PROGRAM F_Gestion_Actionneurs
VAR
	V3V_Bat_Froid_CTA		: Servomoteur_V1;
	Batterie_Elec_CTA		: BatElec;
	Humidificateur			: Humidificateur;
	F_Humi: REAL;
	EF_Humi: BOOL;
	F_BatElec: REAL;
	EF_BatElec: BOOL;
END_VAR
VAR // added by the converter: edge detectors and wires of the graphical bodies
    _w1, _w2 : BOOL;
END_VAR

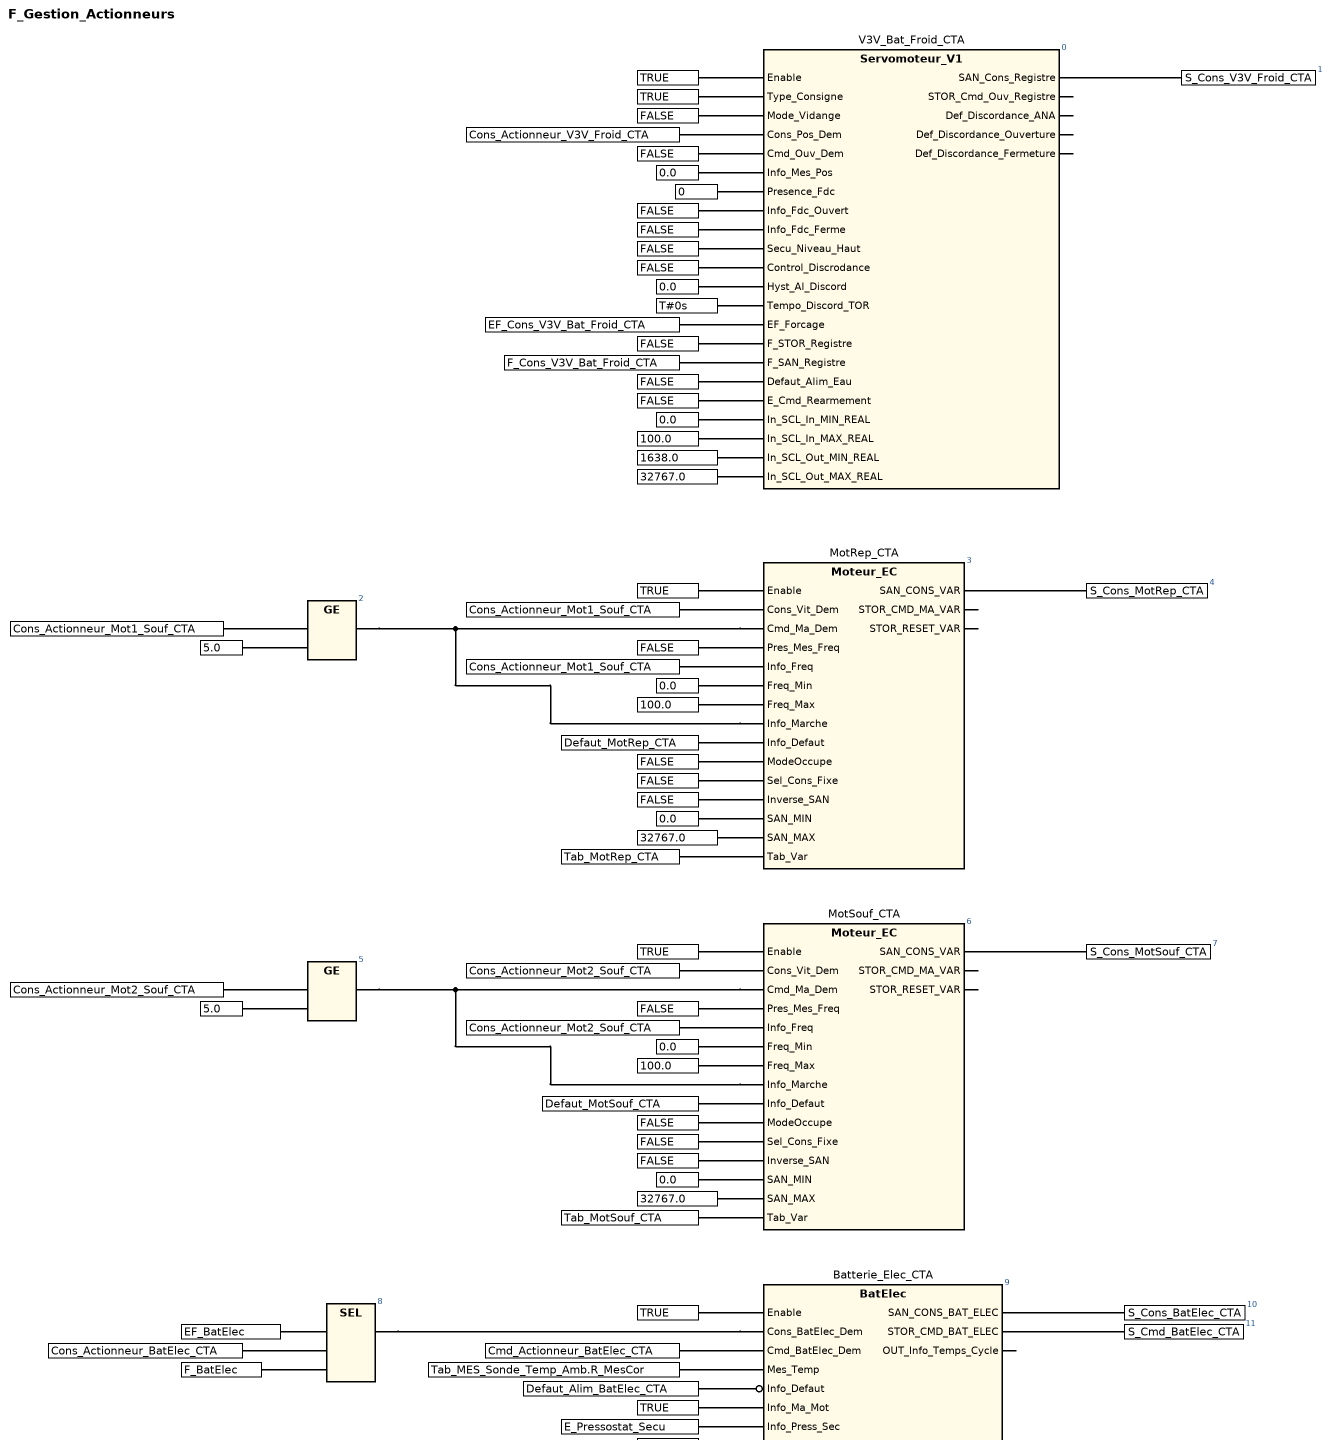
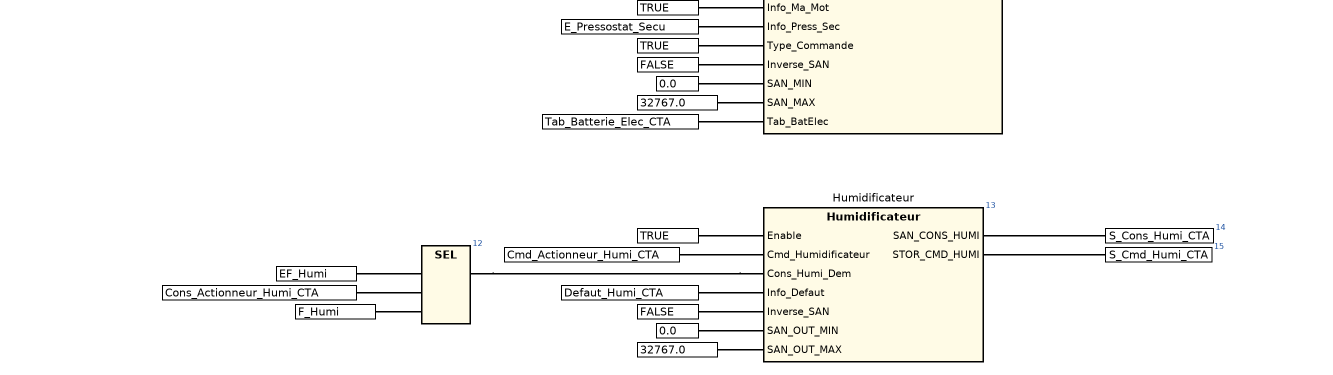
V3V_Bat_Froid_CTA(
    Enable := TRUE,
    Type_Consigne := TRUE,
    Mode_Vidange := FALSE,
    Cons_Pos_Dem := Cons_Actionneur_V3V_Froid_CTA,
    Cmd_Ouv_Dem := FALSE,
    Info_Mes_Pos := 0.0,
    Presence_Fdc := 0,
    Info_Fdc_Ouvert := FALSE,
    Info_Fdc_Ferme := FALSE,
    Secu_Niveau_Haut := FALSE,
    Control_Discrodance := FALSE,
    Hyst_Al_Discord := 0.0,
    Tempo_Discord_TOR := T#0s,
    EF_Forcage := EF_Cons_V3V_Bat_Froid_CTA,
    F_STOR_Registre := FALSE,
    F_SAN_Registre := F_Cons_V3V_Bat_Froid_CTA,
    Defaut_Alim_Eau := FALSE,
    E_Cmd_Rearmement := FALSE,
    In_SCL_In_MIN_REAL := 0.0,
    In_SCL_In_MAX_REAL := 100.0,
    In_SCL_Out_MIN_REAL := 1638.0,
    In_SCL_Out_MAX_REAL := 32767.0); // Servomoteur_V1
S_Cons_V3V_Froid_CTA := V3V_Bat_Froid_CTA.SAN_Cons_Registre;
_w1 := Cons_Actionneur_Mot1_Souf_CTA >= 5.0;
MotRep_CTA(
    Enable := TRUE,
    Cons_Vit_Dem := Cons_Actionneur_Mot1_Souf_CTA,
    Cmd_Ma_Dem := _w1,
    Pres_Mes_Freq := FALSE,
    Info_Freq := Cons_Actionneur_Mot1_Souf_CTA,
    Freq_Min := 0.0,
    Freq_Max := 100.0,
    Info_Marche := _w1,
    Info_Defaut := Defaut_MotRep_CTA,
    ModeOccupe := FALSE,
    Sel_Cons_Fixe := FALSE,
    Inverse_SAN := FALSE,
    SAN_MIN := 0.0,
    SAN_MAX := 32767.0,
    Tab_Var := Tab_MotRep_CTA); // Moteur_EC
S_Cons_MotRep_CTA := MotRep_CTA.SAN_CONS_VAR;
_w2 := Cons_Actionneur_Mot2_Souf_CTA >= 5.0;
MotSouf_CTA(
    Enable := TRUE,
    Cons_Vit_Dem := Cons_Actionneur_Mot2_Souf_CTA,
    Cmd_Ma_Dem := _w2,
    Pres_Mes_Freq := FALSE,
    Info_Freq := Cons_Actionneur_Mot2_Souf_CTA,
    Freq_Min := 0.0,
    Freq_Max := 100.0,
    Info_Marche := _w2,
    Info_Defaut := Defaut_MotSouf_CTA,
    ModeOccupe := FALSE,
    Sel_Cons_Fixe := FALSE,
    Inverse_SAN := FALSE,
    SAN_MIN := 0.0,
    SAN_MAX := 32767.0,
    Tab_Var := Tab_MotSouf_CTA); // Moteur_EC
S_Cons_MotSouf_CTA := MotSouf_CTA.SAN_CONS_VAR;
Batterie_Elec_CTA(
    Enable := TRUE,
    Cons_BatElec_Dem := SEL(EF_BatElec, Cons_Actionneur_BatElec_CTA, F_BatElec),
    Cmd_BatElec_Dem := Cmd_Actionneur_BatElec_CTA,
    Mes_Temp := Tab_MES_Sonde_Temp_Amb.R_MesCor,
    Info_Defaut := NOT Defaut_Alim_BatElec_CTA,
    Info_Ma_Mot := TRUE,
    Info_Press_Sec := E_Pressostat_Secu,
    Type_Commande := TRUE,
    Inverse_SAN := FALSE,
    SAN_MIN := 0.0,
    SAN_MAX := 32767.0,
    Tab_BatElec := Tab_Batterie_Elec_CTA); // BatElec
S_Cons_BatElec_CTA := Batterie_Elec_CTA.SAN_CONS_BAT_ELEC;
S_Cmd_BatElec_CTA := Batterie_Elec_CTA.STOR_CMD_BAT_ELEC;
Humidificateur(
    Enable := TRUE,
    Cmd_Humidificateur := Cmd_Actionneur_Humi_CTA,
    Cons_Humi_Dem := SEL(EF_Humi, Cons_Actionneur_Humi_CTA, F_Humi),
    Info_Defaut := Defaut_Humi_CTA,
    Inverse_SAN := FALSE,
    SAN_OUT_MIN := 0.0,
    SAN_OUT_MAX := 32767.0);
S_Cons_Humi_CTA := Humidificateur.SAN_CONS_HUMI;
S_Cmd_Humi_CTA := Humidificateur.STOR_CMD_HUMI;

END_PROGRAM

(* stored: Version 1.1.0.1, ProductVersion 3.1.4024.12
   POU F_Gestion_Actionneurs: Id {fa7cec6e-9132-4640-a70f-3492371ed5d1}, SpecialFunc None *)
